(* CODESYS project SMC.library
   Company: Ziga Javornik
   DefaultNamespace: ZigaLibs.SMC
   Version: 0.0.3.0
   Placeholder: ZigaLibs.SMC
   Author: Ziga Javornik
   Description: SMC library collection
   Title: ZigaLibs.SMC

Project tree, tasks and I/O mapping:
  libraries: Tc2_Standard, * (Beckhoff Automation GmbH); Tc2_System, * (Beckhoff Automation GmbH); Tc3_Module, * (Beckhoff Automation GmbH); TcUnit, 1.3.1 (www.tcunit.org); ZigaLibs.Core, 0.0.3.7 (Ziga Javornik); ZigaLibs.IoLink, 0.0.0.1 (Ziga Javornik); ZigaLibs.Logging, 0.0.4.1 (Ziga Javornik)
  GVLs/
  SOURCE/
    Flow controllers/
      PFCA7/
        DUTs/
          data type E_PFCA7_AcuumulationShutOff
          data type E_PFCA7_Diagnostic
          data type E_PFCA7_Error
          data type E_PFCA7_FixedOutput
          data type E_PFCA7_FlowRateUnit
          data type E_PFCA7_LocalInput
          data type E_PFCA7_ReferenceCondition
          data type ST_PFCA7_InputProcessData
          data type ST_PFCA7_OutputProcessData
        POUs/
          function block FB_PFCA7 [ST]: FB_init, Execute, Feedback, IoLinkMaxFlowValue, MaxFlow, MeasuredFlow
          interface I_PFCA7: Execute, Feedback, IoLinkMaxFlowValue, MaxFlow, MeasuredFlow
    JXCE1/
      DUTs/
        Aliases/
          data type T_JXCE1_AccDec
          data type T_JXCE1_Force
          data type T_JXCE1_Position
          data type T_JXCE1_Speed
        Commands/
          data type E_JXCE1_MovementMode
          data type ST_JXCE1_Commands
          data type ST_JXCE1_MovementData
          data type ST_JXCE1_NumericalData
        Constants/
          global variables Parameters_JXCE1
        PDO mapping/
          data type ST_JXCE_TxPDO
          data type ST_JXCE1_RxPDO
        Status/
          data type E_JXCE1_AlarmCode
          data type ST_JXCE1_Status
          data type ST_JXE1_MovementFeedback
        data type E_JXCE1_GenericErrors
        data type E_JXCE1_ModeOfOperation
        data type E_JXCE1_State
      POUs/
        function block FB_JXCE1_StepperMotorControl [ST]: ControllerState, Enable, FB_init, Hold, JogBwd, JogFwd, ModeOfOperation, MovementData, MoveToPosition, Reset, ReturnToOrigin, Status, StrokeLength
        interface I_JXCE1_StepperMotorControl: ControllerState, Enable, Hold, JogBwd, JogFwd, ModeOfOperation, MovementData, MoveToPosition, Reset, ReturnToOrigin, Status, StrokeLength
        program JXCE1_Helper [ST]: GetControllerState
    Valve blocks/
      MEC1/
        DUTs/
        POUs/
        data type T_EX260MEC1_ValveList
  TESTS/
    Test suites/
      function block FB_PFCA7_Tests [ST]: Test01_FlowScaling, Test02_FlowLimiting
      function block FB_SUT_Tests [ST]: TestXX_Template
    program PRG_TESTS [ST]
*)

// SOURCE/Flow controllers/PFCA7/DUTs/E_PFCA7_AcuumulationShutOff
{attribute 'qualified_only'}
TYPE E_PFCA7_AcuumulationShutOff :
(
	ShutOffHasNotOccured := 0,
	ShutOffOccured	:= 1
);
END_TYPE

// SOURCE/Flow controllers/PFCA7/DUTs/E_PFCA7_Diagnostic
{attribute 'qualified_only'}
TYPE E_PFCA7_Diagnostic :
(
	WithinRange := 0,
	OutOfRange	:= 1
);
END_TYPE

// SOURCE/Flow controllers/PFCA7/DUTs/E_PFCA7_Error
{attribute 'qualified_only'}
TYPE E_PFCA7_Error :
(
	ErrorNotGenerated := 0,
	ErrorGenerated := 1
);
END_TYPE

// SOURCE/Flow controllers/PFCA7/DUTs/E_PFCA7_FixedOutput
{attribute 'qualified_only'}
TYPE E_PFCA7_FixedOutput :
(
	NormalOutput := 0,
	FixedOutput := 1
);
END_TYPE

// SOURCE/Flow controllers/PFCA7/DUTs/E_PFCA7_FlowRateUnit
{attribute 'qualified_only'}
TYPE E_PFCA7_FlowRateUnit :
(
	Liters := 0,
	CubicFeet := 1
)SINT;
END_TYPE

// SOURCE/Flow controllers/PFCA7/DUTs/E_PFCA7_LocalInput
{attribute 'qualified_only'}
TYPE E_PFCA7_LocalInput :
(
	Remote := 0,
	Local := 1
);
END_TYPE

// SOURCE/Flow controllers/PFCA7/DUTs/E_PFCA7_ReferenceCondition
{attribute 'qualified_only'}
TYPE E_PFCA7_ReferenceCondition :
(
	STD := 0,
	NOR := 1
);
END_TYPE

// SOURCE/Flow controllers/PFCA7/DUTs/ST_PFCA7_InputProcessData
TYPE ST_PFCA7_InputProcessData :
STRUCT
	AccumulatedFlow		: UDINT;
	MeasuredFlow		: INT;
	AC_Error			: BIT;
	FlowError			: BIT;
	PD_OutputError		: BIT;
	AutoShift			: BIT;
	ControlSelect		: BIT;
	FixedOutput			: BIT;
	Error				: BIT;
	SystemError			: BIT;
	OUT_AC				: BIT;
	OUT_Tolerance		: BIT;
	FlowUnit			: E_PFCA7_FlowRateUnit;
	STD_NOT				: BIT;
	
END_STRUCT
END_TYPE

// SOURCE/Flow controllers/PFCA7/DUTs/ST_PFCA7_OutputProcessData
TYPE ST_PFCA7_OutputProcessData :
STRUCT
	CommandedFlowRate	: UINT;
END_STRUCT
END_TYPE

// SOURCE/JXCE1/DUTs/Aliases/T_JXCE1_AccDec
TYPE T_JXCE1_AccDec : REAL; END_TYPE

// SOURCE/JXCE1/DUTs/Aliases/T_JXCE1_Force
TYPE T_JXCE1_Force : UINT(Parameters_JXCE1.PUSHING_FORCE_MIN..Parameters_JXCE1.PUSHING_FORCE_MAX); END_TYPE

// SOURCE/JXCE1/DUTs/Aliases/T_JXCE1_Position
TYPE T_JXCE1_Position : REAL; END_TYPE

// SOURCE/JXCE1/DUTs/Aliases/T_JXCE1_Speed
TYPE T_JXCE1_Speed : REAL; END_TYPE

// SOURCE/JXCE1/DUTs/Commands/E_JXCE1_MovementMode
{attribute 'qualified_only'}
TYPE E_JXCE1_MovementMode :
(
	ABSOLUTE := 1,
	INCREMENTAL := 2
);
END_TYPE

// SOURCE/JXCE1/DUTs/Commands/ST_JXCE1_Commands
TYPE ST_JXCE1_Commands :
STRUCT
	StepData		: ARRAY[0..5] OF BOOL;
	Hold			: BOOL;
	Enable			: BOOL;	// SVON
	SendStepData	: BOOL;	// DRIVE
	Reset			: BOOL;
	ReturnToOrigin	: BOOL;	// SETUP
	JogBackward		: BOOL;
	JogForward		: BOOL;
	FLGHT			: BOOL;
	NumericalData	: ST_JXCE1_NumericalData;
	StartFlag		: BOOL;
	MovementData	: ST_JXCE1_MovementData;
END_STRUCT
END_TYPE

// SOURCE/JXCE1/DUTs/Commands/ST_JXCE1_MovementData
TYPE ST_JXCE1_MovementData :
STRUCT
	MovementMode	: E_JXCE1_MovementMode := E_JXCE1_MovementMode.ABSOLUTE;
	Speed			: T_JXCE1_Speed;
	TargetPosition	: T_JXCE1_Position;
	Acceleration	: T_JXCE1_AccDec;
	Deceleration	: T_JXCE1_AccDec;
	PushingForce	: T_JXCE1_Force;
	TriggerLV		: UINT;
	PushingSpeed	: T_JXCE1_Speed;
	MovingForce		: T_JXCE1_Force;
	AREA1			: T_JXCE1_Position;
	AREA2			: T_JXCE1_Position;
	InPosition		: T_JXCE1_Position;
END_STRUCT
END_TYPE

// SOURCE/JXCE1/DUTs/Commands/ST_JXCE1_NumericalData
TYPE ST_JXCE1_NumericalData :
STRUCT
	SpeedRestriction	: BOOL;
	MovementMode		: BOOL;
	Speed				: BOOL;
	Position			: BOOL;
	Acceleration		: BOOL;
	Deceleration		: BOOL;
	PushingForce		: BOOL;
	TriggerLV			: BOOL;
	PushingSpeed		: BOOL;
	MovingForce			: BOOL;
	AREA1				: BOOL;
	AREA2				: BOOL;
	InPosition			: BOOL;
END_STRUCT
END_TYPE

// SOURCE/JXCE1/DUTs/PDO mapping/ST_JXCE_TxPDO
TYPE ST_JXCE_TxPDO :
STRUCT
	SignalAllocatedToInputPort	: WORD;
	ControllerInformationFlag	: WORD;
	CurrentPosition				: DINT;
	CurrentSpeed				: WORD;
	CurrentPushingForce			: WORD;
	TargetPosition				: DINT;
	Alarm_1						: BYTE;
	Alarm_2						: BYTE;
	Alarm_3						: BYTE;
	Alarm_4						: BYTE;
END_STRUCT
END_TYPE

// SOURCE/JXCE1/DUTs/PDO mapping/ST_JXCE1_RxPDO
TYPE ST_JXCE1_RxPDO :
STRUCT
	OutputPortSignalsAreAllocated	: WORD;
	NumericalDataFlag				: WORD;
	StartFlag                       : BYTE;
	MovementMode                    : BYTE;
	Speed                           : WORD;
	TargetPosition                  : DINT;
	Acceleration                    : WORD;
	Deceleration                    : WORD;
	PushingForce                    : WORD;
	TriggerLV                       : WORD;
	PushingSpeed                    : WORD;
	MovingForce                     : WORD;
	Area1                           : DINT;
	Area2                           : DINT;
	InPosition                      : DINT;
END_STRUCT
END_TYPE

// SOURCE/JXCE1/DUTs/Status/E_JXCE1_AlarmCode
{attribute 'qualified_only'}
//{attribute 'strict'}
{attribute 'to_string'}
TYPE E_JXCE1_AlarmCode :
(
	STEP_DATA_ALM1	:= 48,
	PARAMETER_ALM := 49,
	STEP_DATA_ALM2 := 51,
	STROKE_LIMIT := 52,
	ALM_3A := 58,
	ALM_3D := 61,
	ALM_3E := 62,
	PUSHING_ALM := 96,
	ORIG_ALM := 97,
	SERVO_OFF_ALM := 98,
	DRIVE_ALM := 99,
	ORIG_SENS_ALM := 103,
	OVER_SPEED := 144,
	OVER_MOTOR_VOLTAGE := 145,
	OVER_TEMP := 146,
	OVER_CONTROL_VOLTAGE_147,
	OVER_LOAD := 148,
	POSITION_FAILED_ALM := 149,
	CTRL_COMM_ALM := 150,
	ENOCDER_ALM := 192,
	POLARITY_NOT_FOUND := 193,
	OVER_CURRENT := 194,
	I_SENS_ALM := 195,
	ERR_OVERFLOW := 196,
	MEMORY_ALM := 197,
	CPU_ERROR := 198
)BYTE;
END_TYPE

// SOURCE/JXCE1/DUTs/Status/ST_JXCE1_Status
TYPE ST_JXCE1_Status :
STRUCT
	(* When the operation is started and DRIVE input is turned
	OFF, the step No. executed by the DRIVE signal will be
	refreshed/updated by the combination of OUT0 to OUT5
	(binary digit).*)
	StepData		: BYTE;
	
	(* This terminal is ON during the movement of the actuator
	(during the positioning operation, etc.). 
	WARNING:
	During the pushing operation without movement (no
	movement but the actuator generating the pushing force),
	BUSY is OFF.*)
	Busy			: BOOL;
	
	(* SVRE:
	When the servo motor is OFF, SVRE is OFF. Turns on when
	the servo motor is ON.*)
	Enabled			: BOOL;
	
	(* SETON:
	When the actuator is in the SETON status (the position
	information is established) after returning to origin, this
	terminal is turned ON.
	When the actuator has not returned to origin, this terminal is
	turned OFF.*)
	SETON	: BOOL;
	
	(* INP:
	The condition when the INP output is ON depends on the actuator action:
	- Return to origin
		After stopping the actuator operation (BUSY output is turned
		OFF), the INP is turned ON when the actuator is within the
		range defined in the origin +/-“Default In position” in the
		basic parameter.
	- During positioning operation
		Turns ON when the current position is within "Step data position +/- positioning range".
	- During pushing operation
		Turns ON when the pushing force exceeds the value set in the step data “Trigger LV”. *)
	Done	: BOOL;
	
	(* When the actuator is within the output range between Area1
	and Area2 in the step data, this terminal will turned ON.
	The area output setting range changes depending on the
	active step data.*)
	InRange_AREA	: BOOL;
	
	(* When the actuator is within the output range between "W area
	1 and W area 2" of basic parameter, this terminal will turn ON.*)
	InRange_WAREA	: BOOL;
	
	(* During activation of Teaching Box stop switch, this terminal is
	ON. During the normal operation, this is OFF. This is synchronized to the EMG stop signal input.*)
	ESTOP	: BOOL;
	
	(* Alarm generated when abnormal conditions occur to the
	actuator or its controlling status. OFF when there are no
	alarms. ON in alarm condition.*)
	Alarm	: BOOL;
	
	(* READY turns ON when no alarm is generated with Servo ON*)
	Ready	: BOOL;
	
	MovementFeedback	: ST_JXE1_MovementFeedback;
	
	Alarm_1	: E_JXCE1_AlarmCode;
	Alarm_2	: E_JXCE1_AlarmCode;
	Alarm_3	: E_JXCE1_AlarmCode;
	Alarm_4	: E_JXCE1_AlarmCode;
END_STRUCT
END_TYPE

// SOURCE/JXCE1/DUTs/Status/ST_JXE1_MovementFeedback
TYPE ST_JXE1_MovementFeedback :
STRUCT
	CurrentPosition		: T_JXCE1_Position;
	CurrentSpeed		: T_JXCE1_Position;
	CurrentPushingForce	: T_JXCE1_Force;
	TargetPosition		: T_JXCE1_Position;
END_STRUCT
END_TYPE

// SOURCE/JXCE1/DUTs/E_JXCE1_GenericErrors
{attribute 'qualified_only'}
{attribute 'strict'}
TYPE E_JXCE1_GenericErrors :
(
	SPEED_SET_TOO_LOW := 1000,
	NEGATIVE_SPEED_USED := 1010,
	SET_POSITION_OUT_OF_STROKE_RANGE := 1100
);
END_TYPE

// SOURCE/JXCE1/DUTs/E_JXCE1_ModeOfOperation
{attribute 'qualified_only'}
{attribute 'strict'}
{attribute 'to_string'}
TYPE E_JXCE1_ModeOfOperation :
(
	NUMERICAL,
	STEP_DATA
);
END_TYPE

// SOURCE/JXCE1/DUTs/E_JXCE1_State
{attribute 'qualified_only'}
{attribute 'strict'}
{attribute 'to_string'}
(*
The enum shows the changes in the output signal with respect to the state of the controller. 
*)
TYPE E_JXCE1_State :
(
	POWER_OFF,	// Controller powered down [SVOFF] with no motion
	POWER_ON_NO_MOTION,	// Controller powered down [SVON] with no motion
	RETURNING_TO_ORIGIN, //During returning to origin 
	AT_ORIGIN_POSITION, // The actuator is at the origin. On completion of [SETUP]
	POSITIONING_OR_PUSHING_ACTIVE, // During movement BY positioning/pushing operation
	HOLD, // The actuator is paused by [HOLD]
	POSITIONING_COMPLETE, // On completion of the positioning operation. 
	PUSHING_COMPLETED, // Stopped due to pushing a workload in pushing operation. 
	PUSHING_STOPPED_NO_WORKLOAD_DETECTED, // Stopped due to no detection of workload during a pushing operation. 
	SERVO_OFF_AFTER_RETURNING_TO_ORIGIN, // Servo is OFF after returning to Origin. 
	EMERGENCY, // EMG signal stop from the CN1 connector after the actuator is at the origin
	STATE_UNKNOWN
);
END_TYPE

// SOURCE/Valve blocks/MEC1/T_EX260MEC1_ValveList
TYPE T_EX260MEC1_ValveList : USINT; END_TYPE

// SOURCE/JXCE1/DUTs/Constants/Parameters_JXCE1
{attribute 'qualified_only'}
VAR_GLOBAL CONSTANT
	PUSHING_FORCE_MAX	: UINT := 100; // Maximum pushing force
	PUSHING_FORCE_MIN	: UINT := 0;	// Minimum pushing force
END_VAR

// SOURCE/Flow controllers/PFCA7/POUs/FB_PFCA7
FUNCTION_BLOCK FB_PFCA7 EXTENDS ZigaLibs_IoLink.FB_IoLinkState IMPLEMENTS I_PFCA7
VAR
	InputProcessData	AT %I* : ST_PFCA7_InputProcessData;
	OutputProcessData	AT %Q* : ST_PFCA7_OutputProcessData;
	_inputProcessData	: ST_PFCA7_InputProcessData;
	_maxFlow			: REAL;
	_measuredFlow		: REAL;
	_IoLinkMaxFlowValue	: INT := 4_000;
END_VAR

METHOD FB_init : BOOL
VAR_INPUT
	bInitRetains : BOOL; // if TRUE, the retain variables are initialized (warm start / cold start)
	bInCopyCode : BOOL;  // if TRUE, the instance afterwards gets moved into the copy code (online change)
	logger		: REFERENCE TO ZigaLibs_Logging.I_Logger;
	fMaxFlow	: REAL;
END_VAR
_maxFlow := fMaxFlow;
END_METHOD

(* Should be called cyclically to execute necesary calls
 This is used instead of FBXXX() -> FBXXX.Execute() and makes the programming more consistent.*)
METHOD Execute
VAR_INPUT
	bEnable			: BOOL;	// Enable flow setting
	fFlowSetpoint	: REAL;	// Flow setpoint
END_VAR
_inputProcessData := InputProcessData;

// Flow measurement
_measuredFlow := _maxFlow * (1.0 * InputProcessData.MeasuredFlow)/INT_TO_REAL(_IoLinkMaxFlowValue);

// Output section
IF bEnable = FALSE OR _maxFlow = 0 THEN
	OutputProcessData.CommandedFlowRate := 0;
ELSE
	OutputProcessData.CommandedFlowRate := REAL_TO_UINT((INT_TO_REAL(_IoLinkMaxFlowValue) * MIN(fFlowSetpoint, _maxFlow)/_maxFlow));
END_IF
END_METHOD

 {attribute 'monitoring' := 'variable'}
// Gets device feedback structure
PROPERTY PUBLIC Feedback : REFERENCE TO ST_PFCA7_InputProcessData
GET
Feedback REF= _inputProcessData;
END_GET
END_PROPERTY

(* Gets or sets the IO link max flow value, this is used for value scaling and should be read from the datasheet.*)
PROPERTY IoLinkMaxFlowValue : INT
GET
IoLinkMaxFlowValue := _IoLinkMaxFlowValue;
END_GET
SET
_IoLinkMaxFlowValue := IoLinkMaxFlowValue;
END_SET
END_PROPERTY

(* Gets or sets the max flow*)
PROPERTY MaxFlow : REAL
GET
MaxFlow := _maxFlow;
END_GET
SET
_maxFlow := MaxFlow;
END_SET
END_PROPERTY

(* Gets the measured flow*)
PROPERTY MeasuredFlow : REAL
GET
MeasuredFlow := _measuredFlow;
END_GET
END_PROPERTY

END_FUNCTION_BLOCK

// SOURCE/Flow controllers/PFCA7/POUs/I_PFCA7
INTERFACE I_PFCA7

(* Should be called cyclically to execute necesary calls
 This is used instead of FBXXX() -> FBXXX.Execute() and makes the programming more consistent.*)
METHOD Execute
VAR_INPUT
	bEnable			: BOOL;	// Enable flow setting
	fFlowSetpoint	: REAL;	// Flow setpoint
END_VAR
END_METHOD

// Gets device feedback structure
PROPERTY PUBLIC Feedback : REFERENCE TO ST_PFCA7_InputProcessData
GET
END_GET
END_PROPERTY

// Gets or sets the IO link max flow value, this is used for value scaling and should be read from the datasheet.
PROPERTY IoLinkMaxFlowValue : INT
GET
END_GET
SET
END_SET
END_PROPERTY

// Gets or sets the max flow
PROPERTY PUBLIC MaxFlow : REAL
GET
END_GET
SET
END_SET
END_PROPERTY

// Gets the measured flow
PROPERTY MeasuredFlow : REAL
GET
END_GET
END_PROPERTY

END_INTERFACE

// SOURCE/JXCE1/POUs/FB_JXCE1_StepperMotorControl
(* Function block for SMC JXCE1 stepper motor control.
Constructor:
(strokeLength := ,
 positionUnit := );
*)
FUNCTION_BLOCK FB_JXCE1_StepperMotorControl EXTENDS FB_ErrorSource IMPLEMENTS I_JXCE1_StepperMotorControl 
VAR
	_status				: ST_JXCE1_Status;
	_commands			: ST_JXCE1_Commands;
	_state				: E_JXCE1_State;
	_resetTimer			: Tc2_Standard.TON := (PT := T#100MS);
	_strokeLength		: REAL;
	_valueFor1mm		: REAL;
	_startFlagDelay		: Tc2_Standard.TOF;
	_modeOfOperation	: E_JXCE1_ModeOfOperation := E_JXCE1_ModeOfOperation.NUMERICAL;
	_minSpeed			: T_JXCE1_Speed;
	_sb					: ZigaLibs_Core.FB_StringBuilder;
END_VAR

VAR
	SendData	AT %Q* 	: ST_JXCE1_RxPDO;
	ReceiveData	AT %I*	: ST_JXCE_TxPDO;
END_VAR

_state := JXCE1_Helper.GetControllerState(controller := THIS^);
_status.StepData.0 := ReceiveData.SignalAllocatedToInputPort.0;
_status.StepData.1 := ReceiveData.SignalAllocatedToInputPort.1;
_status.StepData.2 := ReceiveData.SignalAllocatedToInputPort.2;
_status.StepData.3 := ReceiveData.SignalAllocatedToInputPort.3;
_status.StepData.4 := ReceiveData.SignalAllocatedToInputPort.4;
_status.StepData.5 := ReceiveData.SignalAllocatedToInputPort.5;

_status.Busy := ReceiveData.SignalAllocatedToInputPort.8;
_status.Enabled := ReceiveData.SignalAllocatedToInputPort.9;
_status.SETON := ReceiveData.SignalAllocatedToInputPort.10;
_status.Done := ReceiveData.SignalAllocatedToInputPort.11;
_status.InRange_AREA := ReceiveData.SignalAllocatedToInputPort.12;
_status.InRange_WAREA := ReceiveData.SignalAllocatedToInputPort.13;
_status.ESTOP := ReceiveData.SignalAllocatedToInputPort.14;
_status.Alarm := ReceiveData.SignalAllocatedToInputPort.15;

IF _status.Alarm THEN
	THIS^.Error := TRUE;
	THIS^.GenericError.Code := TO_DINT(_status.Alarm_1);
	THIS^.GenericError.Message := _sb.Reset()
		.AddString('Driver alarm active: ')
		.AddWithDblQuotationMarks(TO_STRING(_status.Alarm_1))
		.Create();
END_IF

_status.Ready := ReceiveData.ControllerInformationFlag.4;
IF _valueFor1mm <> 0 THEN
	_status.MovementFeedback.CurrentPosition := DINT_TO_REAL(ReceiveData.CurrentPosition) * _valueFor1mm;
END_IF

_status.MovementFeedback.CurrentSpeed := WORD_TO_REAL(ReceiveData.CurrentSpeed);
_status.MovementFeedback.CurrentPushingForce := WORD_TO_UINT(ReceiveData.CurrentPushingForce);
IF _valueFor1mm <> 0 THEN
	_status.MovementFeedback.TargetPosition := DINT_TO_REAL(ReceiveData.TargetPosition) * _valueFor1mm;	
END_IF

_status.Alarm_1 := ReceiveData.Alarm_1;
_status.Alarm_2 := ReceiveData.Alarm_2;
_status.Alarm_3 := ReceiveData.Alarm_3;
_status.Alarm_4 := ReceiveData.Alarm_4;

IF NOT _commands.Enable THEN
	_commands.SendStepData := FALSE;
	_commands.ReturnToOrigin := FALSE;
END_IF

_resetTimer(IN := _commands.Reset);
IF _resetTimer.Q THEN
	_commands.Reset := FALSE;
END_IF

IF (_status.SETON AND _status.Done) OR _state = E_JXCE1_State.SERVO_OFF_AFTER_RETURNING_TO_ORIGIN THEN
	_commands.ReturnToOrigin := FALSE;
END_IF

// Step data
SendData.OutputPortSignalsAreAllocated.0 := _commands.StepData[0] AND _modeOfOperation = E_JXCE1_ModeOfOperation.STEP_DATA;
SendData.OutputPortSignalsAreAllocated.1 := _commands.StepData[1] AND _modeOfOperation = E_JXCE1_ModeOfOperation.STEP_DATA;
SendData.OutputPortSignalsAreAllocated.2 := _commands.StepData[2] AND _modeOfOperation = E_JXCE1_ModeOfOperation.STEP_DATA;
SendData.OutputPortSignalsAreAllocated.3 := _commands.StepData[3] AND _modeOfOperation = E_JXCE1_ModeOfOperation.STEP_DATA;
SendData.OutputPortSignalsAreAllocated.4 := _commands.StepData[4] AND _modeOfOperation = E_JXCE1_ModeOfOperation.STEP_DATA;
SendData.OutputPortSignalsAreAllocated.5 := _commands.StepData[5] AND _modeOfOperation = E_JXCE1_ModeOfOperation.STEP_DATA;
SendData.OutputPortSignalsAreAllocated.6 := FALSE;
SendData.OutputPortSignalsAreAllocated.7 := FALSE;

// Commands
SendData.OutputPortSignalsAreAllocated.8 := _commands.Hold;
SendData.OutputPortSignalsAreAllocated.9 := _commands.Enable;
SendData.OutputPortSignalsAreAllocated.10 := _commands.SendStepData;
SendData.OutputPortSignalsAreAllocated.11 := _commands.Reset;
SendData.OutputPortSignalsAreAllocated.12 := _commands.ReturnToOrigin;
SendData.OutputPortSignalsAreAllocated.13 := _commands.JogBackward;
SendData.OutputPortSignalsAreAllocated.14 := _commands.JogForward;

// Method calling to jog - reset every body call
_commands.JogBackward := FALSE;
_commands.JogForward := FALSE;

SendData.OutputPortSignalsAreAllocated.15 := _commands.FLGHT;

// Numerical mode - enable sending of all parameters when in this mode
SendData.NumericalDataFlag.0 := FALSE;
SendData.NumericalDataFlag.1 := FALSE;//_modeOfOperation = E_JXCE1_ModeOfOperation.NUMERICAL AND NOT _commands.ReturnToOrigin;
SendData.NumericalDataFlag.2 := FALSE;
SendData.NumericalDataFlag.3 := FALSE;
SendData.NumericalDataFlag.4 := _modeOfOperation = E_jxce1_modeOfOperation.NUMERICAL AND NOT _commands.ReturnToOrigin;
SendData.NumericalDataFlag.5 := _modeOfOperation = E_jxce1_modeOfOperation.NUMERICAL AND NOT _commands.ReturnToOrigin;
SendData.NumericalDataFlag.6 := _modeOfOperation = E_jxce1_modeOfOperation.NUMERICAL AND NOT _commands.ReturnToOrigin;
SendData.NumericalDataFlag.7 := _modeOfOperation = E_jxce1_modeOfOperation.NUMERICAL AND NOT _commands.ReturnToOrigin;
SendData.NumericalDataFlag.8 := _modeOfOperation = E_jxce1_modeOfOperation.NUMERICAL AND NOT _commands.ReturnToOrigin;
SendData.NumericalDataFlag.9 := _modeOfOperation = E_jxce1_modeOfOperation.NUMERICAL AND NOT _commands.ReturnToOrigin;
SendData.NumericalDataFlag.10 := _modeOfOperation = E_jxce1_modeOfOperation.NUMERICAL AND NOT _commands.ReturnToOrigin;
SendData.NumericalDataFlag.11 := _modeOfOperation = E_jxce1_modeOfOperation.NUMERICAL AND NOT _commands.ReturnToOrigin;
SendData.NumericalDataFlag.12 := _modeOfOperation = E_jxce1_modeOfOperation.NUMERICAL AND NOT _commands.ReturnToOrigin;
SendData.NumericalDataFlag.13 := _modeOfOperation = E_jxce1_modeOfOperation.NUMERICAL AND NOT _commands.ReturnToOrigin;
SendData.NumericalDataFlag.14 := _modeOfOperation = E_jxce1_modeOfOperation.NUMERICAL AND NOT _commands.ReturnToOrigin;
SendData.NumericalDataFlag.15 := _modeOfOperation = E_jxce1_modeOfOperation.NUMERICAL AND NOT _commands.ReturnToOrigin;


SendData.StartFlag.0 := _commands.StartFlag;
SendData.MovementMode := TO_BYTE(_commands.MovementData.MovementMode);
SendData.Speed := REAL_TO_UINT(_commands.MovementData.Speed);
IF _valueFor1mm <> 0 THEN
	SendData.TargetPosition := REAL_TO_DINT(_commands.MovementData.TargetPosition / _valueFor1mm);
END_IF
SendData.Acceleration := REAL_TO_UINT(_commands.MovementData.Acceleration);
SendData.Deceleration := REAL_TO_UINT(_commands.MovementData.Deceleration);
SendData.PushingForce := _commands.MovementData.PushingForce;
SendData.TriggerLV := _commands.MovementData.TriggerLV;
SendData.PushingSpeed := REAL_TO_UINT(_commands.MovementData.PushingSpeed);
SendData.MovingForce := _commands.MovementData.MovingForce;
IF _valueFor1mm <> 0 THEN
	SendData.Area1 := REAL_TO_DINT(_commands.MovementData.AREA1 / _valueFor1mm);
	SendData.Area2 := REAL_TO_DINT(_commands.MovementData.AREA2 / _valueFor1mm);
	SendData.InPosition := REAL_TO_DINT(_commands.MovementData.InPosition / _valueFor1mm);	
END_IF

// Start flag in method calling, reset every call in case the method is not called any more
_commands.StartFlag := FALSE;

{attribute 'monitoring':='variable'}
(* Gets the controller state*)
PROPERTY ControllerState : E_JXCE1_State
GET
ControllerState := _state;
END_GET
END_PROPERTY

{attribute 'monitoring':='variable'}
(* Enables or disables the controller*)
PROPERTY Enable : BOOL
GET
Enable := _commands.Enable;
END_GET
SET
_commands.Enable := Enable;
END_SET
END_PROPERTY

METHOD FB_init : BOOL
VAR_INPUT
	bInitRetains 	: BOOL; // if TRUE, the retain variables are initialized (warm start / cold start)
	bInCopyCode 	: BOOL;  // if TRUE, the instance afterwards gets moved into the copy code (online change)
	strokeLength	: T_JXCE1_Position;	// Stroke length in mm
	valueFor1mm		: T_JXCE1_Position;	// Defines how many units are required for a mm. Example : 10 = provided position of 1 is equal to 0.1mm
	minSpeed		: T_JXCE1_Speed;
END_VAR
_strokeLength := strokeLength;
_valueFor1mm := valueFor1mm;
_minSpeed := minSpeed;
END_METHOD

{attribute 'monitoring':='variable'}
(* If set to TRUE, axis is halted with maximum deceleration*)
PROPERTY Hold : BOOL
GET
Hold := _commands.Hold;
END_GET
SET
_commands.Hold := Hold;
END_SET
END_PROPERTY

(* Jogs backward with the defined speed*)
METHOD JogBwd
_commands.JogBackward := TRUE;
END_METHOD

(* Jogs forward with the defined speed*)
METHOD JogFwd
_commands.JogForward := TRUE;
END_METHOD

{attribute 'monitoring':='variable'}
(* Gets or sets the mode of operation for the unit*)
PROPERTY ModeOfOperation : E_JXCE1_ModeOfOperation
GET
ModeOfOperation := _modeOfOperation;
END_GET
SET
_modeOfOperation := ModeOfOperation;
END_SET
END_PROPERTY

{attribute 'monitoring':='variable'}
(* Gets or sets various movement data properties*)
PROPERTY MovementData : REFERENCE TO ST_JXCE1_MovementData
GET
MovementData REF= _commands.MovementData;
END_GET
SET
_commands.MovementData := MovementData;
END_SET
END_PROPERTY

(* Moves to the target position with the defined speed. Returns TRUE when done*)
METHOD MoveToPosition : BOOL
VAR_INPUT
	speed		: T_JXCE1_Speed;	// Speed in mm/s
	position	: T_JXCE1_Position;	// Position in mm
END_VAR

VAR_OUTPUT
	error		: BOOL; // If incorrect parameters are used error will be TRUE
	errorInfo	: ZigaLibs_Core.ST_GenericError;	// Error information can be found in this struct
END_VAR

VAR_INST
	Rtrig_Done			: Tc2_Standard.R_TRIG;
END_VAR

VAR
	targetSpeed	: T_JXCE1_Speed;
	sb			: ZigaLibs_Core.FB_StringBuilder;
	stErrorInfo	: ZigaLibs_Core.ST_GenericError;
END_VAR
Rtrig_Done(CLK := _status.Done AND _status.SETON AND _status.Ready AND NOT _status.Busy);
error := FALSE;

IF speed < _minSpeed THEN
	stErrorInfo.Code := E_JXCE1_GenericErrors.SPEED_SET_TOO_LOW;
	stErrorInfo.Message := sb.AddString('Speed setpoint too low!')
		.AddString('Set speed: ').AddAnyReal(speed, 2, FALSE).AddString('mm/s. ')
		.AddString('Minimum allowed speed is ').AddAnyReal(_minSpeed, 2 , FALSE).AddString('mm/s.')
		.Create();
	error := TRUE;
	errorInfo := stErrorInfo;
	RETURN;
END_IF

IF speed < 0 THEN
	stErrorInfo.Code := E_JXCE1_GenericErrors.NEGATIVE_SPEED_USED;
	stErrorInfo.Message := sb.AddString('Negative speed not allowed!').Create();
	error := TRUE;
	errorInfo := stErrorInfo;
	RETURN;
END_IF

IF (_commands.MovementData.MovementMode = E_JXCE1_MovementMode.ABSOLUTE AND (position > _strokeLength)) OR
   (_commands.MovementData.MovementMode = E_JXCE1_MovementMode.INCREMENTAL AND ((position + _status.MovementFeedback.CurrentPosition) > _strokeLength))
THEN
	stErrorInfo.Code := E_JXCE1_GenericErrors.SET_POSITION_OUT_OF_STROKE_RANGE;
	stErrorInfo.Message := sb.AddString('Target position would result in out of stroke range movement!')
		.AddString('Position setpoint: ').AddAnyReal(position, 2, FALSE).AddString('mm')
		.AddString(', movement mode used: ').AddWithDblQuotationMarks(TO_STRING(_commands.MovementData.MovementMode))
		.Create();
		
	error := TRUE;
	errorInfo := stErrorInfo;
	RETURN;
END_IF

// If done, start flag will not be sent - new method call starts new positioning command
IF Rtrig_Done.Q THEN
	MoveToPosition := TRUE;
	RETURN;
END_IF

targetSpeed := speed;
_commands.StartFlag := TRUE;
_commands.MovementData.PushingForce := 0;
_commands.MovementData.TargetPosition := position;
_commands.MovementData.Speed := speed;
END_METHOD

{warning 'add method implementation '}
(* Resets the controller when called*)
METHOD Reset
_commands.Reset := TRUE;
_commands.ReturnToOrigin := FALSE;
THIS^.ResetError();
END_METHOD

(* Returns axis to origin*)
METHOD ReturnToOrigin
_commands.ReturnToOrigin := TRUE;
END_METHOD

{attribute 'monitoring':='variable'}
(* Gets the controller status structure*)
PROPERTY Status : REFERENCE TO ST_JXCE1_Status
GET
Status REF= _status;
END_GET
END_PROPERTY

{attribute 'monitoring':='variable'}
// Gets the stroke length (mm) of the actuator
PROPERTY StrokeLength : REAL
GET
StrokeLength := _strokeLength;
END_GET
END_PROPERTY

END_FUNCTION_BLOCK

// SOURCE/JXCE1/POUs/JXCE1_Helper
{attribute 'no_explicit_call' := 'Body contains no logic, calling methods only allowed.'}
PROGRAM JXCE1_Helper
VAR
END_VAR

// Returns the controller state based on various signals of the controller
METHOD GetControllerState	: E_JXCE1_State
VAR_INPUT
	controller	: I_JXCE1_StepperMotorControl;
END_VAR
IF  NOT controller.Status.Busy AND
	NOT controller.Status.Done AND
	NOT controller.Status.Enabled AND
	NOT controller.Status.SETON AND
	controller.Status.StepData = 0 
THEN
	GetControllerState := E_JXCE1_State.POWER_OFF;
	RETURN;
END_IF

IF  NOT controller.Status.Busy AND
	NOT controller.Status.Done AND
	controller.Status.Enabled AND
	NOT controller.Status.SETON AND
	controller.Status.StepData = 0 
THEN
	GetControllerState := E_JXCE1_State.POWER_ON_NO_MOTION;
	RETURN;
END_IF

IF  controller.Status.Busy AND
	NOT controller.Status.Done AND
	controller.Status.Enabled AND
	NOT controller.Status.SETON AND
	controller.Status.StepData = 0 
THEN
	GetControllerState := E_JXCE1_State.RETURNING_TO_ORIGIN;
	RETURN;
END_IF

IF  NOT controller.Status.Busy AND
	controller.Status.Done AND
	controller.Status.Enabled AND
	controller.Status.SETON AND
	controller.Status.StepData = 0 
THEN
	GetControllerState := E_JXCE1_State.AT_ORIGIN_POSITION;
	RETURN;
END_IF

IF  controller.Status.Busy AND
	NOT controller.Status.Done AND
	controller.Status.Enabled AND
	controller.Status.SETON AND
	controller.Status.StepData <> 0 {warning 'preveri, ne vem vrednosti...'}
THEN
	GetControllerState := E_JXCE1_State.POSITIONING_OR_PUSHING_ACTIVE;
	RETURN;
END_IF

IF  NOT controller.Status.Busy AND
	NOT controller.Status.Done AND
	controller.Status.Enabled AND
	controller.Status.SETON AND
	controller.Status.StepData <> 0 {warning 'preveri, ne vem vrednosti...'}
THEN
	GetControllerState := E_JXCE1_State.HOLD;
	RETURN;
END_IF

IF  NOT controller.Status.Busy AND
	controller.Status.Done AND
	controller.Status.Enabled AND
	controller.Status.SETON AND
	controller.Status.StepData <> 0 {warning 'preveri, ne vem vrednosti...'}
THEN
	GetControllerState := E_JXCE1_State.POSITIONING_COMPLETE;
	RETURN;
END_IF

IF  NOT controller.Status.Busy AND
	controller.Status.Done AND
	controller.Status.Enabled AND
	controller.Status.SETON AND
	controller.Status.StepData <> 0 {warning 'preveri, ne vem vrednosti...'}
THEN
	GetControllerState := E_JXCE1_State.PUSHING_COMPLETED;
	RETURN;
END_IF

IF  NOT controller.Status.Busy AND
	NOT controller.Status.Done AND
	controller.Status.Enabled AND
	controller.Status.SETON AND
	controller.Status.StepData = 0
THEN
	GetControllerState := E_JXCE1_State.PUSHING_STOPPED_NO_WORKLOAD_DETECTED;
	RETURN;
END_IF

IF  NOT controller.Status.Busy AND
	NOT controller.Status.Done AND
	NOT controller.Status.Enabled AND
	controller.Status.SETON AND
	controller.Status.StepData <> 0 {warning 'preveri, ne vem vrednosti...'}
THEN
	GetControllerState := E_JXCE1_State.SERVO_OFF_AFTER_RETURNING_TO_ORIGIN;
	RETURN;
END_IF

IF  NOT controller.Status.Busy AND
	NOT controller.Status.Done AND
	NOT controller.Status.Enabled AND
	controller.Status.SETON AND
	controller.Status.StepData = 0
THEN
	GetControllerState := E_JXCE1_State.EMERGENCY;
	RETURN;
END_IF
END_METHOD

END_PROGRAM

// SOURCE/JXCE1/POUs/I_JXCE1_StepperMotorControl
INTERFACE I_JXCE1_StepperMotorControl

// Gets the controller state
PROPERTY ControllerState : E_JXCE1_State
GET
END_GET
END_PROPERTY

// Enables or disables the controller
PROPERTY Enable : BOOL
GET
END_GET
SET
END_SET
END_PROPERTY

// Gets or sets whether the axis is haleted
PROPERTY Hold : BOOL
GET
END_GET
SET
END_SET
END_PROPERTY

// Jogs backward with the defined speed
METHOD JogBwd
END_METHOD

// Jogs forward with the defined speed
METHOD JogFwd
END_METHOD

// Gets or sets the mode of operation for the unit
PROPERTY ModeOfOperation : E_JXCE1_ModeOfOperation
GET
END_GET
SET
END_SET
END_PROPERTY

// Gets or sets various movement data properties
PROPERTY MovementData : REFERENCE TO ST_JXCE1_MovementData
GET
END_GET
SET
END_SET
END_PROPERTY

// Moves to the target position with the defined speed. Returns TRUE when done
METHOD MoveToPosition : BOOL
VAR_INPUT
	speed		: T_JXCE1_Speed;	// Speed in mm/s
	position	: T_JXCE1_Position;	// Position in mm
END_VAR

VAR_OUTPUT
	error		: BOOL; // If incorrect parameters are used error will be TRUE
	errorInfo	: ZigaLibs_Core.ST_GenericError;	// Error information can be found in this struct
END_VAR
END_METHOD

// Resets the controller when called
METHOD Reset
END_METHOD

// Returns axis to origin
METHOD ReturnToOrigin
END_METHOD

// Gets the controller status structure
PROPERTY Status : REFERENCE TO ST_JXCE1_Status
GET
END_GET
END_PROPERTY

// Gets the stroke length (mm) of the actuator
PROPERTY StrokeLength : REAL
GET
END_GET
END_PROPERTY

END_INTERFACE

// TESTS/Test suites/FB_PFCA7_Tests
// A collection of tests for PFCA7 SMC series
FUNCTION_BLOCK INTERNAL FB_PFCA7_Tests EXTENDS FB_TestSuite
VAR_INPUT
END_VAR
VAR_OUTPUT
END_VAR
VAR
		_maxProcessDataFlowSetpoint : UINT := 4000;
END_VAR

Test01_FlowScaling();
Test02_FlowLimiting();

METHOD PRIVATE Test01_FlowScaling
VAR_INST
	fbFlowController_100slm	: FB_PFCA7(logger := 0, fMaxFlow := 100.0);
	fbFlowController_50slm	: FB_PFCA7(logger := 0, fMaxFlow := 50.0);
END_VAR
TcUnit.TEST('Test01_FlowScaling');

fbFlowController_100slm.Execute(bEnable := TRUE, fFlowSetpoint := 0);
fbFlowController_50slm.Execute(bEnable := TRUE, fFlowSetpoint := 0);
AssertEquals_REAL(
	Actual := fbFlowController_100slm.OutputProcessData.CommandedFlowRate,
	Expected := 0.0,
	Delta := 0,
	Message := 'Incorrect commanded flow setpoint when setting flow to 0!');
AssertEquals(
	Actual := fbFlowController_100slm.OutputProcessData.CommandedFlowRate,
	Expected := fbFlowController_50slm.OutputProcessData.CommandedFlowRate,
	Message := 'Flow setpoint for 100 and 50 slm flow controller differs!');
	

fbFlowController_100slm.Execute(bEnable := TRUE, fFlowSetpoint := 50.0);
AssertEquals_REAL(
	Actual := fbFlowController_100slm.OutputProcessData.CommandedFlowRate,
	Expected := 2000.0,
	Delta := 0.1,
	Message := 'Incorrect commanded flow setpoint when setting flow to 50!');

fbFlowController_100slm.Execute(bEnable := TRUE, fFlowSetpoint := 100.0);
fbFlowController_50slm.Execute(bEnable := TRUE, fFlowSetpoint := 50.0);
AssertEquals(
	Actual := fbFlowController_100slm.OutputProcessData.CommandedFlowRate,
	Expected := _maxProcessDataFlowSetpoint,
	Message := 'Incorrect commanded flow setpoint when setting flow to 100!');

AssertEquals(
	Actual := fbFlowController_100slm.OutputProcessData.CommandedFlowRate,
	Expected := fbFlowController_50slm.OutputProcessData.CommandedFlowRate,
	Message := 'Flow setpoint for 100 and 50 slm flow controller differs!');
	
TcUnit.TEST_FINISHED();
END_METHOD

METHOD PRIVATE Test02_FlowLimiting
VAR_INST
	fbFlowController_100slm	: FB_PFCA7(logger := 0, fMaxFlow := 100.0);
	fbFlowController_50slm	: FB_PFCA7(logger := 0, fMaxFlow := 50.0);
END_VAR
TcUnit.TEST('Test02_FlowLimiting');

fbFlowController_100slm.Execute(bEnable := TRUE, fFlowSetpoint := 200.0);

AssertEquals(
	Expected := _maxProcessDataFlowSetpoint,
	Actual := fbFlowController_100slm.OutputProcessData.CommandedFlowRate,
	Message := 'Flow should not exceed the maximum set value!');

fbFlowController_100slm.MaxFlow := 30.0;
AssertEquals(
	Expected := _maxProcessDataFlowSetpoint,
	Actual := fbFlowController_100slm.OutputProcessData.CommandedFlowRate,
	Message := 'Max flow setting should not be exceeded after changing the value of the upper limit!!');	
	
TcUnit.TEST_FINISHED();
END_METHOD

END_FUNCTION_BLOCK

// TESTS/Test suites/FB_SUT_Tests
// Subject under test
FUNCTION_BLOCK INTERNAL FB_SUT_Tests EXTENDS FB_TestSuite

// Create instance variables that will be accesible for all tests
VAR
	fbLinearMotor	: FB_JXCE1_StepperMotorControl(
		strokeLength := 50.0,
 		valueFor1mm := 0.01,
		minSpeed	:= 0);
END_VAR

// Call your test methods here
TestXX_Template();

METHOD PRIVATE TestXX_Template

(* Instanced variables are VERY useful for writing tests since tests are run in paralel (by default).
By instantiating local variables that are not placed on the same stack as method (values are retained between calls)
you make sure that the SUT is not changed by some other test. *)
VAR_INST
	
END_VAR

// Place temporary variables here
VAR
	
END_VAR
// The name of the test, is the same as method name!
// Use this for paralel unit tests
// TcUnit.TEST('TestXX_Template');

// Use this for running tests in sequence
IF TcUnit.TEST_ORDERED('TestXX_Template') THEN
	// Do your assertions here...
	AssertTrue(
		Condition := FALSE, 
		Message := 'Implement tests!');

	TcUnit.TEST_FINISHED();
END_IF
END_METHOD

END_FUNCTION_BLOCK

// TESTS/PRG_TESTS
PROGRAM INTERNAL PRG_TESTS

(* Instantiate test suites here. Naming convention for tests should be a suffix with _Tests.
Good practice for creating test methods is to end them with _test as well. *)
VAR
	PFCA7_Tests	: FB_PFCA7_Tests;
END_VAR

// Run tests in parallel
//TcUnit.RUN();

// Run tests in sequence, one after the other.
TcUnit.RUN_IN_SEQUENCE();

END_PROGRAM
